// TIA Portal V20 export
VAR_GLOBAL   // PLC tag table "mission_Robot"
END_VAR
VAR_GLOBAL CONSTANT   // user constants
   MISSION_ExtractTray : Int := 202;
   MISSION_Load_Pallet : Int := 300;   // carico pallet a seguito di comando HMI
   MISSION_LoadGripper : Int := 220;
   MISSION_LoadManVice : Int := 140;
   MISSION_LoadPallet_MC : Int := 100;
   MISSION_LoadPart_MC : Int := 120;
   MISSION_LoadPartOnRobot : Int := 200;
   MISSION_ReleaseTray : Int := 203;
   MISSION_Unload_Pallet : Int := 301;   // scarico pallet a seguito di comando HMI
   MISSION_UnloadGripper : Int := 210;
   MISSION_UnloadManVice : Int := 150;
   MISSION_UnloadPallet_MC : Int := 110;
   MISSION_UnloadPart_MC : Int := 130;
   MISSION_UnloadPartFromRobot : Int := 201;
   MISSION_SwapGripper : Int := 230;
   MISSION_PickPart_TRAY_HMI : Int := 211;
   MISSION_PlacePart_TRAY_HMI : Int := 212;
   MISSION_PickPart_MC_HMI : Int := 213;
   MISSION_PlacePart_MC_HMI : Int := 214;
   MISSION_PickPallet_MC_HMI : Int := 215;
   MISSION_PlacePallet_MC_HMI : Int := 216;
   MISSION_OpenGripper1 : Int := 240;
   MISSION_CloseGripper1 : Int := 241;
   MISSION_OpenGripper2 : Int := 242;
   MISSION_CloseGripper2 : Int := 243;
   MISSION_PickPlacePart_MC : Int := 135;
   MISSION_PositioningMC_AUTO : Int := 145;
   MISSION_RobotHome_AUTO : Int := 146;
END_VAR
